// TIA Portal V20 export
DATA_BLOCK "QDAS_ReceiveRelation"   // DB300
{ S7_Optimized_Access := 'TRUE' }
// stored: MemoryReserve 100
   VAR
      processData : Bool;
      spareOut_1 : Bool;
      spareOut_2 : Bool;
      spareOut_3 : Bool;
      spareOut_4 : Bool;
      spareOut_5 : Bool;
      spareOut_6 : Bool;
      spareOut_7 : Bool;
      "type" : Int;
      module : Int;
      machine : DInt;
      fixture : Int;
      pun : Array[0..31] of Char;
      unWinderInfeed : Struct
         "Unwind Tension Set Point 1" : Real;
         "Unwind Tension Actual 1" : Real;
         "Unwind Roll Diameter 1" : Real;
         "Unwind Roll Diameter 2" : Real;
         "Bobbin ID 1" : String;
         "Bobbin ID 2" : String;
         "Cycle end Trigger" : Bool;
         Blocked : Bool;
         Starved : Bool;
         "Good Count" : DInt;
         "Reject Count" : DInt;
         "Fault bit" : Bool;
         Fault : Bool;
         PUN : String;
         "Part Type" : String;
         "FTQ & Reject code" : String;
      END_STRUCT;
      reelCutInspection : Struct
         "Introcut count 1" : DInt;
         "Introcut Vision - Tab length 1" : Real;
         "Introcut Vision - Tab height 1" : Real;
         "Introcut Vision - Electrode length 1" : Real;
         "Introcut Vision - Electrode height 1" : Real;
         "Introcut Vision - Gap between left edge & Tab 1" : Real;
         "Introcut Vision - Gap between tab & right edge 1" : Real;
         "Introcut Vision - Height of Ceramic Coating" : Real;
         "Introcut Vision - Radii 1" : Real;
         "Introcut Vision - Height (y) of total electrode (ini. Tab) 1" : Real;
         "OK/NG" : String;
         "Cycle end Trigger" : Bool;
         Blocked : Bool;
         Starved : Bool;
         "Good Count" : DInt;
         "Reject Count" : DInt;
         "Fault bit" : Bool;
         Fault : Bool;
         PUN : String;
         "FTQ & Reject code" : String;
         "Target Cycle Time" : String;
         "Material Low" : DInt;
         "2d Matrix" : String;
         "Tool Change" : DInt;
      END_STRUCT;
   END_VAR
BEGIN
END_DATA_BLOCK
